ABB RAPID module: CalibData.modx

MODULE CalibData
    PERS tooldata tVacuum:=[TRUE,[[0,0,150],[1,0,0,0]],[1,[0,0,1],[1,0,0,0],0,0,0]];
ENDMODULE
